{attribute addProperty BoxType "EL5101-0010-0016"}
{attribute addProperty Id "StatusAT %I*Status_F1BDA5E31621Counter_valueAT %I*UINT16217Latch_valueAT %I*UINT16218"}
{attribute addProperty CRC "3195579534"}
{attribute addProperty SizeInBites "48"}
{attribute addProperty SizeInBytes "6"}
TYPE ENC_Status_compact_BE78AC8E :
STRUCT
	{attribute addProperty Name "Status"}
	Status AT %I* : Status_F1BDA5E3;
	{attribute addProperty Name "Counter_value"}
	Counter_value AT %I* : UINT;
	{attribute addProperty Name "Latch_value"}
	Latch_value AT %I* : UINT;
END_STRUCT
END_TYPE

(* stored: Version 1.2.0.0, ProductVersion 3.1.4024.9
   DUT ENC_Status_compact_BE78AC8E: Id {2697eaf6-635d-45ec-9cb5-dbe4983c9e95} *)
